ABB RobotStudio station: SD_RStudioExe02_240523.rsstnx

Station SD_RStudioExe02_240523 (saved by RobotStudio 22.3.10190.2)
Controller CRB15000_5_95
  mechanical unit ROB_1: CRB15000_5_95__02, 6 joints, base frame (0, 0, 0) mm
Layout (positions relative to the parent item):
  - CRB15000_5_95__02 [mechanism, from Robots\CRB15000_5_95__02.rslib] at (0, 0, 0) mm; joint values [-0.145, 0.728, -0.9691, 0.6517, 1.503, -1.2291] (rad or m)
  - MyTool [mechanism, from Training Objects\myTool.rslib] at (827.48, -62.38, 762.56) mm, rotated rx -174.22 ry 40.71 rz -112.35 deg
  - Curve_thing [part, from Training Objects\Curve_Thing.rslib] at (759.86, -58.9, 454.67) mm, rotated rx 0 ry -5.23 rz 7.04 deg
Attachment: MyTool is attached to CRB15000_5_95__02 / Link6
Attachment: wbj_part is attached to Curve_thing
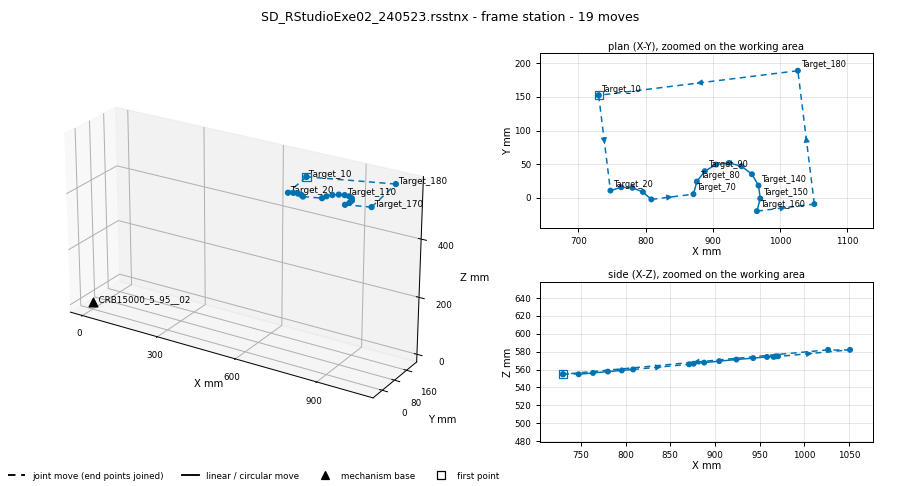
[picture p0: tool path of SD_RStudioExe02_240523.rsstnx in frame station, 19 of 19 moves have a stored position in this frame; points joined in program order, loops and branches not executed]
Targets, tools, work objects and paths stored in the station, written as RAPID:
! task T_ROB1
MODULE CalibData
  PERS tooldata MyTool:=[TRUE,[[31.792631019,0,229.638935148],[0.945518576,0,0.325568154,0]],[1,[0,0,1],[1,0,0,0],0,0,0]];
  PERS wobjdata wbj_part:=[FALSE,TRUE,"",[[751.723,-59.909,544.3],[0.997073284,0.002800799,-0.045502576,0.061372121]],[[0,0,0],[1,0,0,0]]];
ENDMODULE

! task T_ROB1
MODULE Module1
  CONST robtarget Target_10:=[[5.447771522,213.325999251,9.999631539],[0.000000274,-0.476687486,0.87907283,-0.000000147],[0,0,0,0],[9E+09,9E+09,9E+09,9E+09,9E+09,9E+09]];
  CONST robtarget Target_20:=[[5.447813914,70.452455009,9.999631179],[0.000000274,-0.476687486,0.87907283,-0.000000147],[0,0,0,0],[9E+09,9E+09,9E+09,9E+09,9E+09,9E+09]];
  CONST robtarget Target_30:=[[22.005959529,73.353353936,9.999641472],[0.000000274,-0.476687486,0.87907283,-0.000000147],[0,0,0,0],[9E+09,9E+09,9E+09,9E+09,9E+09,9E+09]];
  CONST robtarget Target_40:=[[38.589703046,70.602562816,9.999651766],[0.000000274,-0.476687486,0.87907283,-0.000000147],[0,0,0,0],[9E+09,9E+09,9E+09,9E+09,9E+09,9E+09]];
  CONST robtarget Target_50:=[[53.324501672,62.511017214,9.999660899],[0.000000274,-0.476687486,0.87907283,-0.000000147],[0,0,0,0],[9E+09,9E+09,9E+09,9E+09,9E+09,9E+09]];
  CONST robtarget Target_60:=[[64.544808032,49.993344666,9.999667836],[0.000000274,-0.476687486,0.87907283,-0.000000147],[0,0,0,0],[9E+09,9E+09,9E+09,9E+09,9E+09,9E+09]];
  CONST robtarget Target_70:=[[127.96500608,49.993363483,9.999707231],[0.000000274,-0.476687486,0.87907283,-0.000000147],[0,0,0,0],[9E+09,9E+09,9E+09,9E+09,9E+09,9E+09]];
  CONST robtarget Target_80:=[[135.282825319,68.050908377,9.999711823],[0.000000274,-0.476687486,0.87907283,-0.000000147],[0,0,0,0],[9E+09,9E+09,9E+09,9E+09,9E+09,9E+09]];
  CONST robtarget Target_90:=[[148.946837819,81.940478865,9.999720346],[0.000000274,-0.476687486,0.87907283,-0.000000147],[0,0,0,0],[9E+09,9E+09,9E+09,9E+09,9E+09,9E+09]];
  CONST robtarget Target_100:=[[166.882161063,89.552941416,9.999731505],[0.000000274,-0.476687486,0.87907283,-0.000000147],[0,0,0,0],[9E+09,9E+09,9E+09,9E+09,9E+09,9E+09]];
  CONST robtarget Target_110:=[[186.365313305,89.732342353,9.999743608],[0.000000274,-0.476687486,0.87907283,-0.000000147],[0,0,0,0],[9E+09,9E+09,9E+09,9E+09,9E+09,9E+09]];
  CONST robtarget Target_120:=[[204.437774712,82.451439617,9.999754815],[0.000000274,-0.476687486,0.87907283,-0.000000147],[0,0,0,0],[9E+09,9E+09,9E+09,9E+09,9E+09,9E+09]];
  CONST robtarget Target_130:=[[218.355239085,68.815839468,9.999763427],[0.000000274,-0.476687486,0.87907283,-0.000000147],[0,0,0,0],[9E+09,9E+09,9E+09,9E+09,9E+09,9E+09]];
  CONST robtarget Target_140:=[[226.004337199,50.896110006,9.999768132],[0.000000274,-0.476687486,0.87907283,-0.000000147],[0,0,0,0],[9E+09,9E+09,9E+09,9E+09,9E+09,9E+09]];
  CONST robtarget Target_150:=[[226.223552263,31.413365057,9.99976822],[0.000000274,-0.476687486,0.87907283,-0.000000147],[0,0,0,0],[9E+09,9E+09,9E+09,9E+09,9E+09,9E+09]];
  CONST robtarget Target_160:=[[218.979596435,13.326062608,9.999763674],[0.000000274,-0.476687486,0.87907283,-0.000000147],[0,0,0,0],[9E+09,9E+09,9E+09,9E+09,9E+09,9E+09]];
  CONST robtarget Target_170:=[[305.447830864,13.326088264,9.999817385],[0.000000274,-0.476687486,0.87907283,-0.000000147],[0,0,0,0],[9E+09,9E+09,9E+09,9E+09,9E+09,9E+09]];
  CONST robtarget Target_180:=[[305.447771522,213.326088263,9.99981789],[0.000000274,-0.476687486,0.87907283,-0.000000147],[0,0,0,0],[9E+09,9E+09,9E+09,9E+09,9E+09,9E+09]];
  CONST robtarget Target_190:=[[5.447771522,213.325999251,9.999631539],[0.000000274,-0.476687486,0.87907283,-0.000000147],[0,0,0,0],[9E+09,9E+09,9E+09,9E+09,9E+09,9E+09]];
  PROC Path_10()
    MoveJ Target_10,v1000,z100,MyTool\WObj:=wbj_part;
    MoveJ Target_20,v1000,z100,MyTool\WObj:=wbj_part;
    MoveL Target_30,v1000,z100,MyTool\WObj:=wbj_part;
    MoveL Target_40,v1000,z100,MyTool\WObj:=wbj_part;
    MoveL Target_50,v1000,z100,MyTool\WObj:=wbj_part;
    MoveL Target_60,v1000,z100,MyTool\WObj:=wbj_part;
    MoveJ Target_70,v1000,z100,MyTool\WObj:=wbj_part;
    MoveL Target_80,v1000,z100,MyTool\WObj:=wbj_part;
    MoveL Target_90,v1000,z100,MyTool\WObj:=wbj_part;
    MoveL Target_100,v1000,z100,MyTool\WObj:=wbj_part;
    MoveL Target_110,v1000,z100,MyTool\WObj:=wbj_part;
    MoveL Target_120,v1000,z100,MyTool\WObj:=wbj_part;
    MoveL Target_130,v1000,z100,MyTool\WObj:=wbj_part;
    MoveL Target_140,v1000,z100,MyTool\WObj:=wbj_part;
    MoveL Target_150,v1000,z100,MyTool\WObj:=wbj_part;
    MoveL Target_160,v1000,z100,MyTool\WObj:=wbj_part;
    MoveJ Target_170,v1000,z100,MyTool\WObj:=wbj_part;
    MoveJ Target_180,v1000,z100,MyTool\WObj:=wbj_part;
    MoveJ Target_190,v1000,z100,MyTool\WObj:=wbj_part;
  ENDPROC
ENDMODULE

